TYPE ST_WaferStatus :
STRUCT
	// Managed by module
	// Non-zero and unique within one Module; array index is storage only.
	EndpointId : UDINT;
	EndpointName : STRING(80);
	MaterialContext : ST_MaterialContext;
END_STRUCT
END_TYPE

(* stored: Version 1.1.0.1, ProductVersion 3.1.4026.18
   DUT ST_WaferStatus: Id {14f9d5f9-39d1-4854-bedd-e4f7b43e695c} *)
